FUNCTION_BLOCK Train2
  (* Standard: 61499-2 *)
  (* Version 0,1, 2015-00-24, Th?o, PC_THEO *)
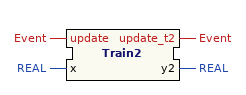
  EVENT_INPUT
    update;
  END_EVENT
  EVENT_OUTPUT
    update_t2;
  END_EVENT
  VAR_INPUT
    x : REAL;
  END_VAR
  VAR_OUTPUT
    y2 : REAL;
  END_VAR
  VAR
    d : REAL;
    k : INT;
    C1y2 : REAL;
    delta : REAL;
  END_VAR
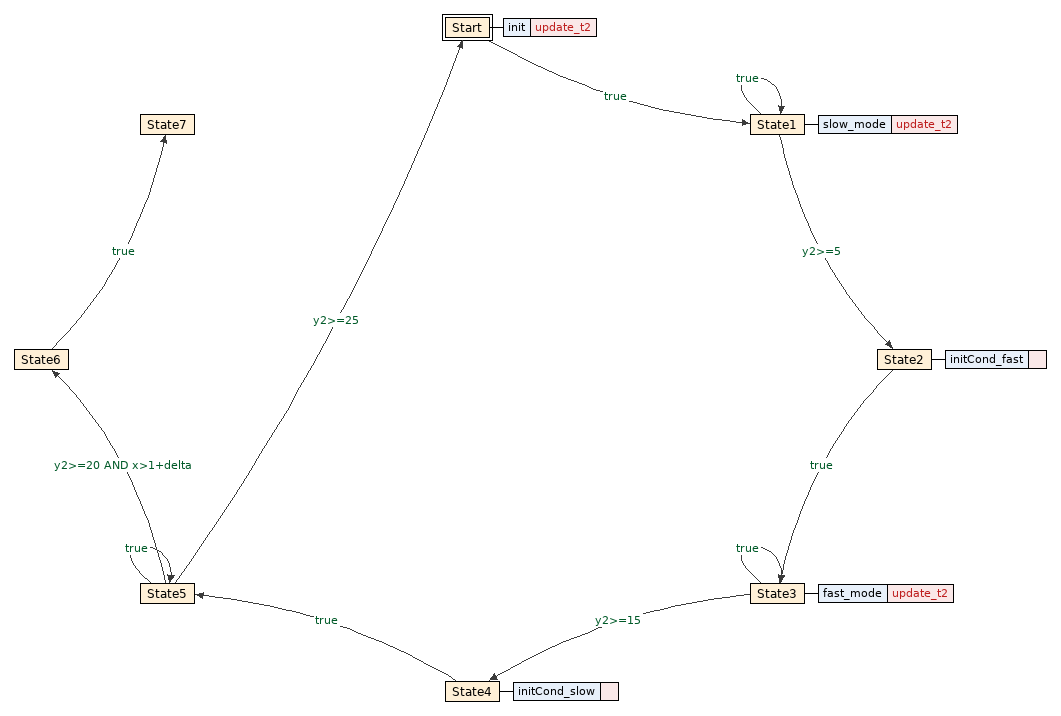
  EC_STATES
    Start : init -> update_t2;
    State1 : slow_mode -> update_t2;
    State2 : initCond_fast;
    State3 : fast_mode -> update_t2;
    State4 : initCond_slow;
    State5;
    State6;
    State7;
  END_STATES
  EC_TRANSITIONS
    Start TO State1 := true;
    State1 TO State2 := y2>=5;
    State1 TO State1 := true;
    State2 TO State3 := true;
    State3 TO State4 := y2>=15;
    State3 TO State3 := true;
    State4 TO State5 := true;
    State5 TO State6 := y2>=20 AND x>1+delta;
    State5 TO Start := y2>=25;
    State5 TO State5 := true;
    State6 TO State7 := true;
  END_TRANSITIONS
  ALGORITHM init IN C:
me->y2=0;
me->delta=0.0001;
me->k=1;
me->C1y2=-1.5;
  END_ALGORITHM
  ALGORITHM slow_mode IN C:
me->y2=me->C1y2*exp(-0.5*me->d*me->k)+1;
(me->k)++;
  END_ALGORITHM
  ALGORITHM fast_mode IN C:
me->y2=me->C1y2*exp(-1.5*me->d*me->k)+3;
(me->k)++;
  END_ALGORITHM
  ALGORITHM emergency_brake IN C:
me->y2=me->C1y2*exp(-1.0L/15.0L*me->d*me->k);
(me->k)++;

if (me->y2 <= me->delta) {
	printf ("Emergency brake : Train stopped at y2 = %f and x = %f\n",me->y2, me->x);
	exit(1);
	}
  END_ALGORITHM
  ALGORITHM initCond_slow IN C:
me->k=1;
me->C1y2=me->x-1.5;
printf("Train 2 is going into slow mode \n");
  END_ALGORITHM
  ALGORITHM initCond_fast IN C:
me->k=1;
me->C1y2=me->x-3;
printf("Train 2 is going into fast mode \n");
  END_ALGORITHM
  ALGORITHM initCond_brake IN C:
me->k=1;
me->C1y2=me->x-15;
printf("Emergency brake T2 !!!\n");
  END_ALGORITHM
END_FUNCTION_BLOCK
